ABB RobotStudio station: medicine_dispatcher_part1.rspag

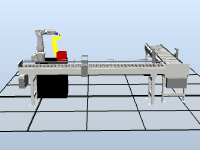
--- station ---
Station proyecto final SFM (saved by RobotStudio 6.8.8307.1040)
Controller IRB_120_3kg_0.58m_2, task T_ROB1: task frame (RAPID world) sits at (0, 0, 794.13) mm in the station
Controller IRB_120_3kg_0.58m_2
  mechanical unit ROB_1: IRB120_3_58__01, 6 joints, base frame (0, 0, 0) mm
Layout (positions relative to the parent item):
  - IRB120_3_58__01 [mechanism, from Robots\IRB120_3_58_G_01.rslib] at (0, 0, 794.13) mm; joint values [-0.0026, 0, 0, 0.0046, 0.5236, -0.0053] (rad or m)
  - MyNewTool [mechanism, from Libraries\chupon.rslib] at (364.35, -0.8, 1388.12) mm, rotated rx -180 ry 60 rz -180 deg
  - Positioner_cubo [smart component, from Components\Positioner.rslib]
      properties: Object=CAJA; Position=[0.285 0.1 0.1008]; Orientation=[0 0 0]; Reference=Global; ReferenceObject=(none)
  - Attacher [smart component, from Components\Attacher.rslib]
      properties: Parent=MyNewTool; Flange=0; Child=CAJA; Mount=false; Offset=[0 0 0]; Orientation=[0 0 0]
  - Detacher [smart component, from Components\Detacher.rslib]
      properties: Child=CAJA; KeepPosition=true
  - CAJA [part] at (62.11, -86.03, 797.36) mm
  - Componente inteligente_1 [smart component]
      signals: DI colsion, DO copia
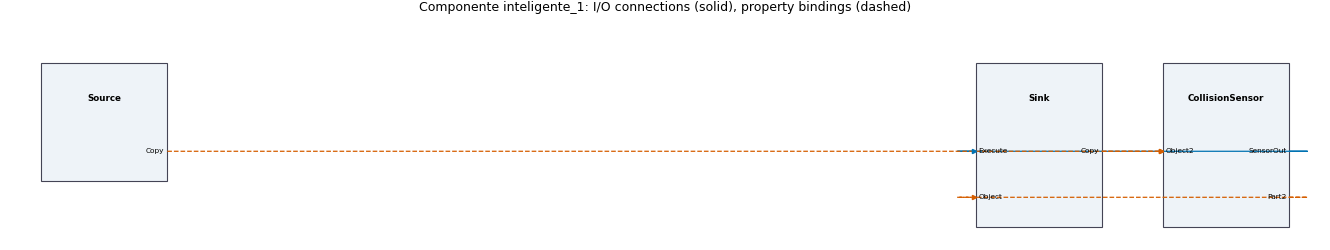
      connections:
        CollisionSensor.SensorOut -> Sink.Execute
        Source.Copy => CollisionSensor.Object2
        CollisionSensor.Part2 => Sink.Object
        Source.Copy => CollisionSensor.Object2
    - cinta [part] at (175.62, 0, 0) mm
    - CollisionSensor [smart component, from Components\CollisionSensor.rslib]
        properties: Object1=cinta2; Object2=(none); NearMiss=0.01; Part1=(none); Part2=(none); CollisionType=0
    - 400_guide [part, from Equipment\Conveyor Guide 400.rslib] at (-361.11, -595.71, 0) mm
    - Source [smart component, from Components\Source.rslib]
        properties: Source=CAJA; Copy=(none); Parent=(none); Position=[0.062111 -0.08603 0.79736]; Orientation=[0 0 0]; Transient=false; PhysicsBehavior=3
  - tope [part] at (-27.41, 42.13, 271.69) mm
  - Pieza_1 [part] at (0, 114.8, 0) mm
  - Pieza_2 [part] at (-99.17, -123.81, 0) mm
  - cinta2 [part, from Equipment\Conveyor Guide 400.rslib] at (3010.82, -631.88, 0) mm, rotated rx 0 ry 0 rz 90 deg
Attachment: MyNewTool is attached to IRB120_3_58__01 / Link6
Station signals: DI posicionador_cubo
Station logic (signal -> signal, property => property):
  proyecto final SFM.posicionador_cubo -> Positioner_cubo.Execute
  IRB_120_3kg_0.58m_2.attach_cubo -> Attacher.Execute
  IRB_120_3kg_0.58m_2.detach_cubo -> Detacher.Execute
Targets, tools, work objects and paths stored in the station and not in the controller backup, written as RAPID:
! task T_ROB1
MODULE Module1
  CONST robtarget Target_10:=[[455.691796359,-0.795818432,541.253938558],[0.5,0,0.866025404,0],[0,0,0,0],[9E+09,9E+09,9E+09,9E+09,9E+09,9E+09]];
  CONST robtarget Target_20:=[[302.000006174,-0.795818432,452.519938558],[0.000000017,0,1,0],[-1,0,-1,0],[9E+09,9E+09,9E+09,9E+09,9E+09,9E+09]];
  CONST robtarget Target_30:=[[349.585716801,4.170948431,199.987938558],[0,1,0,0],[0,0,2,0],[9E+09,9E+09,9E+09,9E+09,9E+09,9E+09]];
  CONST robtarget Target_40:=[[347.286720378,-362.351627791,185.269742824],[0,1,0,0],[-1,0,1,0],[9E+09,9E+09,9E+09,9E+09,9E+09,9E+09]];
  CONST robtarget Target_40_2:=[[291.184201422,-216.512339255,495.782245252],[0,1,0,0],[-1,0,1,0],[9E+09,9E+09,9E+09,9E+09,9E+09,9E+09]];
  CONST robtarget Target_10_2:=[[455.691796359,-0.795818432,541.253938558],[0.5,0,0.866025404,0],[-1,0,-1,0],[9E+09,9E+09,9E+09,9E+09,9E+09,9E+09]];
  CONST robtarget Target_30_2_2:=[[289.448,22.770378063,562.155341196],[0,1,0,0],[0,0,2,0],[9E+09,9E+09,9E+09,9E+09,9E+09,9E+09]];
  CONST robtarget Target_10_3:=[[455.691796359,-0.795818432,541.253938558],[0.5,0,0.866025404,0],[0,0,0,0],[9E+09,9E+09,9E+09,9E+09,9E+09,9E+09]];
  PROC Path_10()
    MoveL Target_10,v1000,z100,MyNewTool\WObj:=wobj0;
    MoveL Target_20,v150,fine,MyNewTool\WObj:=wobj0;
    MoveL Target_30,v150,fine,MyNewTool\WObj:=wobj0;
    PulseDO attach_cubo;
    WaitTime 1;
    MoveL Target_30_2_2,v1000,z100,MyNewTool\WObj:=wobj0;
    MoveL Target_40,v150,fine,MyNewTool\WObj:=wobj0;
    PulseDO detach_cubo;
    WaitTime 1;
    MoveL Target_40_2,v150,fine,MyNewTool\WObj:=wobj0;
    WaitTime 1;
    MoveL Target_10_2,v1000,z100,MyNewTool\WObj:=wobj0;
    WaitTime 1;
  ENDPROC
ENDMODULE


--- Backups/IRB_120_3kg_0.58m_2/RAPID/TASK1/PROGMOD/CalibData.mod ---
MODULE CalibData
	PERS tooldata MyNewTool:=[TRUE,[[0,0,105.468],[1,0,0,0]],[1,[0,0,1],[1,0,0,0],0,0,0]];
ENDMODULE

--- Backups/IRB_120_3kg_0.58m_2/SYSPAR/EIO.cfg ---
EIO:CFG_1.0:6:1::
#
INDUSTRIAL_NETWORK:

      -Name "DeviceNet" -Label "DeviceNet Master/Slave Network" -Address "2"
#
DEVICENET_INTERNAL_DEVICE:

      -Name "DN_Internal_Device" -VendorName "ABB Robotics"\
      -ProductName "DeviceNet Internal Slave Device"
#
EIO_SIGNAL:

      -Name "attach_cubo" -SignalType "DO"

      -Name "detach_cubo" -SignalType "DO"
